FUNCTION_BLOCK FB_Roboter_E
VAR_INPUT
END_VAR
VAR_OUTPUT
END_VAR
VAR
END_VAR

END_FUNCTION_BLOCK

(* stored: Version 1.1.0.1, ProductVersion 3.1.4024.15
   POU FB_Roboter_E: Id {4af811a2-b766-4668-b73b-cadf1a937bf2}, SpecialFunc None *)
